TYPE ST_MoverState :
STRUCT
	bInPlacePosition			: BOOL; 	//Wózek w pozycji wyjmowania zamknięć	
	bPlaceAllowed				: BOOL;		//Zezwolenie na pobranie nasadki
	bInPickPosition				: BOOL; 	//Wózek w pozycjach wkładania zamknięć
	bMovingInPickPos			: BOOL;		//Wózek przemieszcza się w pozycji Pick 
	bWaitingForGoToPickPosition	: BOOL;		//Wózek czeka na przejscie do pick w biezpiecznej pozycji 
	bSlot1InPlacePosition		: BOOL;		//Gniazdo 1 ustawione w pozycji wkładania zamknięć
	bSlot2InPlacePosition		: BOOL;		//Gniazdo 2 ustawione w pozycji wkładania zamknięć
	bSlot3InPlacePosition		: BOOL;		//Gniazdo 3 ustawione w pozycji wkładania zamknięć
	bSlot4InPlacePosition		: BOOL;		//Gniazdo 4 ustawione w pozycji wkładania zamknięć
	stSlotStatus				: ARRAY [1..4] OF ST_SlotStatus;		//Gniazdo zapełnione
	bEmpty						: BOOL;		//Pusty wózek
	bFull						: BOOL; 	//zapełniony wózek
	iSlotNo						: INT;		//Nr gniazda
END_STRUCT
END_TYPE

(* stored: Version 1.2.0.0, ProductVersion 3.1.4026.13, FileIdentifier fd0522889678605a894f428ef2d85ddd6944c2a6, FileSignature 315c916ca81fbcef70d4bccfc80c312d40039c6f60a560e2283455b86b69916ce9fe7bd1d8e22d342a3496be9fefe511fc9c7ce9f0acd2d698a21e36e9f981a259d8d35f6d12f46228d555dfe6c058abdfa7bf1a8968012194d93338e7fc1f9c17e46b63c312616330b2f039348e7f3dc54d1ca362f2b2b77bcb5d0069cc2bafd9513433009155daf2021da5d482969ffc3cc76c1e2b36b81b386b9ca856946eda0df23b6eb9c83526ccbc67e9645b0da20275ea2d3b7a9749868187aaf3c03dc805ae1a25daf79542e2bc9fe2715269611498e6b7a649f7e323d2da516a55d17c505cf0d7c4c69395d88933d93a1c8a38df9b11472428f87690d3f166d99ca3
   DUT ST_MoverState: Id {db0177f3-65af-4bc6-9e56-66607c782b31} *)
